/// each unit can run in its own PROGRAM and Task, respectively. However, this is optional and one may also
/// instantiate the unit in the ModuleProgram.
/// In order to keep initialization to a minimum, all ModuleContext objects that are required by the Unit are
/// given as FB_init parameter. These objects are
/// * data structs
/// * communication structs
/// * busmaster(s)
/// A unit should always be a root object (no parent) if it is running in its own context. If it runs in the same
/// task as the Module the parent may be set to the Module's Application.
PROGRAM MachineUnitProgram
VAR
{region "Machine"}
{undefine RunInSeparateProgram}
{IF NOT (defined (Machine_disabled)) AND (defined (RunInSeparateProgram))}
  Machine : MachineUnit(name := 'Machine', // name of the unit (for logging)
					  parent := 0, // caller of the Unit's cyclic method. If the Unit runs in its own context use 0
						configdata := ZGlobal.Data.Config.Machine,
						machinedata := ZGlobal.Data.Machine.Machine,
						calibrationdata := ZGlobal.Data.Calibration.Machine,
						com := ZGlobal.Com.Unit.Machine);
  {attribute 'section' := '__ZwPlcUnitProgramDeclaration__'}
  {attribute 'ZId' := 'ffcc16ae-32b8-4aad-8514-f391c00062a3'}
{END_IF}
{endregion}
{attribute '__ZwPlcUnitProgramDeclaration__'} // Do not remove this attribute! It is used for code generation.
END_VAR

// run the unit - the cylics of all children will be called as well

{region "Machine"}
{undefine RunInSeparateProgram}
{IF NOT (defined (Machine_disabled)) AND (defined (RunInSeparateProgram))}
  Machine.Cyclic();
  {attribute 'section' := '__ZwPlcUnitProgramImplementation__'}
  {attribute 'ZId' := 'ffcc16ae-32b8-4aad-8514-f391c00062a3'}
{END_IF}
{endregion}
{attribute '__ZwPlcUnitProgramImplementation__'} // Do not remove this attribute! It is used for code generation.

END_PROGRAM

(* stored: Version 1.1.0.1
   POU MachineUnitProgram: Id {fc5ce30b-e02b-4862-a1d4-d9c4155c9471}, SpecialFunc None *)
